Fanuc TP program (LS listing): KAREL_CONTROL.LS

/PROG  KAREL_CONTROL
/ATTR
OWNER		= MNEDITOR;
COMMENT		= "";
PROG_SIZE	= 185;
CREATE		= DATE 22-07-08  TIME 10:50:56;
MODIFIED	= DATE 22-07-08  TIME 13:44:02;
FILE_NAME	= ;
VERSION		= 0;
LINE_COUNT	= 1;
MEMORY_SIZE	= 561;
PROTECT		= READ_WRITE;
TCD:  STACK_SIZE	= 0,
      TASK_PRIORITY	= 50,
      TIME_SLICE	= 0,
      BUSY_LAMP_OFF	= 0,
      ABORT_REQUEST	= 0,
      PAUSE_REQUEST	= 0;
DEFAULT_GROUP	= *,*,*,*,*;
CONTROL_CODE	= 00000000 00000000;
LOCAL_REGISTERS	= 0,0,0;
/APPL

LINE_TRACK;
  LINE_TRACK_SCHEDULE_NUMBER      : 0;
  LINE_TRACK_BOUNDARY_NUMBER      : 0;
  CONTINUE_TRACK_AT_PROG_END      : TRUE;

/MN
   1:  RUN DATA_INPUT ;
/POS
/END
